// TIA Portal V17 export
// export: Created 2025-03-05T07:59:13.1679611Z, ExportSetting WithDefaults, DisplayName Totally Integrated Automation Portal, DisplayVersion V17 Update 8, DisplayName TIA Portal Openness, DisplayVersion V17 Update 8, DisplayName TIA Portal Version Control Interface, DisplayVersion V17, DisplayName SINAMICS Startdrive Advanced, DisplayVersion V17 SP2, DisplayName SINAMICS Startdrive G110M, G120, G120C, G120D, G120P, G115D, DisplayVersion V17 SP2, DisplayName SINAMICS Startdrive G130, G150, S120, S150, SINAMICS MV, S210, DisplayVersion V17 SP2, DisplayName STEP 7 Professional, DisplayVersion V17 Update 8, DisplayName SINUMERIK ONE STEP 7 Toolbox, DisplayVersion V17 Update 12, DisplayName SINUMERIK 840D sl STEP 7 Toolbox, DisplayVersion V17 Update 12, DisplayName STEP 7 Safety, DisplayVersion V17 Update 6, DisplayName WinCC Advanced, DisplayVersion V17 Update 8
FUNCTION "FC4001_FIXTURES_CALIBRATION" : Void   // FC4001, LAD
{ S7_Optimized_Access := 'TRUE' }
VERSION : 0.1
// stored: AutoNumber false, IsIECCheckEnabled false, SetENOAutomatically false, UDAEnableTagReadback false
BEGIN

REGION Network 1: FIXTURE 1 STATION 2 CALIBRATION DONE MEMORY
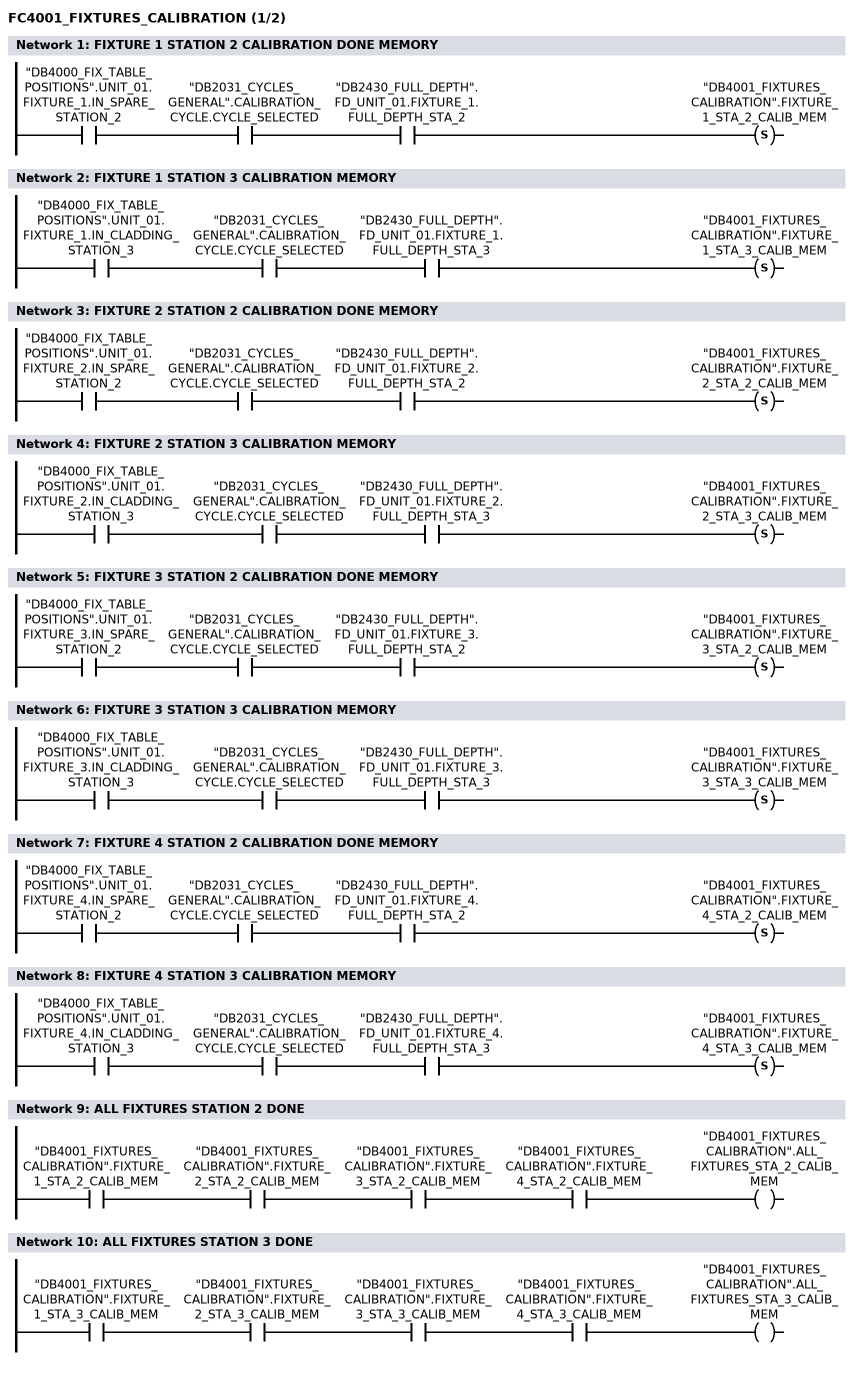
   RUNG wire#powerrail
      Contact( "DB4000_FIX_TABLE_POSITIONS".UNIT_01.FIXTURE_1.IN_SPARE_STATION_2 )
      Contact( "DB2031_CYCLES_GENERAL".CALIBRATION_CYCLE.CYCLE_SELECTED )
      Contact( "DB2430_FULL_DEPTH".FD_UNIT_01.FIXTURE_1.FULL_DEPTH_STA_2 )
      S_Coil( "DB4001_FIXTURES_CALIBRATION".FIXTURE_1_STA_2_CALIB_MEM )
   END_RUNG
   // the same network as SCL:
   IF "DB4000_FIX_TABLE_POSITIONS".UNIT_01.FIXTURE_1.IN_SPARE_STATION_2 AND "DB2031_CYCLES_GENERAL".CALIBRATION_CYCLE.CYCLE_SELECTED AND "DB2430_FULL_DEPTH".FD_UNIT_01.FIXTURE_1.FULL_DEPTH_STA_2 THEN
       "DB4001_FIXTURES_CALIBRATION".FIXTURE_1_STA_2_CALIB_MEM := TRUE;
   END_IF;
END_REGION

REGION Network 2: FIXTURE 1 STATION 3 CALIBRATION MEMORY
   RUNG wire#powerrail
      Contact( "DB4000_FIX_TABLE_POSITIONS".UNIT_01.FIXTURE_1.IN_CLADDING_STATION_3 )
      Contact( "DB2031_CYCLES_GENERAL".CALIBRATION_CYCLE.CYCLE_SELECTED )
      Contact( "DB2430_FULL_DEPTH".FD_UNIT_01.FIXTURE_1.FULL_DEPTH_STA_3 )
      S_Coil( "DB4001_FIXTURES_CALIBRATION".FIXTURE_1_STA_3_CALIB_MEM )
   END_RUNG
   // the same network as SCL:
   IF "DB4000_FIX_TABLE_POSITIONS".UNIT_01.FIXTURE_1.IN_CLADDING_STATION_3 AND "DB2031_CYCLES_GENERAL".CALIBRATION_CYCLE.CYCLE_SELECTED AND "DB2430_FULL_DEPTH".FD_UNIT_01.FIXTURE_1.FULL_DEPTH_STA_3 THEN
       "DB4001_FIXTURES_CALIBRATION".FIXTURE_1_STA_3_CALIB_MEM := TRUE;
   END_IF;
END_REGION

REGION Network 3: FIXTURE 2 STATION 2 CALIBRATION DONE MEMORY
   RUNG wire#powerrail
      Contact( "DB4000_FIX_TABLE_POSITIONS".UNIT_01.FIXTURE_2.IN_SPARE_STATION_2 )
      Contact( "DB2031_CYCLES_GENERAL".CALIBRATION_CYCLE.CYCLE_SELECTED )
      Contact( "DB2430_FULL_DEPTH".FD_UNIT_01.FIXTURE_2.FULL_DEPTH_STA_2 )
      S_Coil( "DB4001_FIXTURES_CALIBRATION".FIXTURE_2_STA_2_CALIB_MEM )
   END_RUNG
   // the same network as SCL:
   IF "DB4000_FIX_TABLE_POSITIONS".UNIT_01.FIXTURE_2.IN_SPARE_STATION_2 AND "DB2031_CYCLES_GENERAL".CALIBRATION_CYCLE.CYCLE_SELECTED AND "DB2430_FULL_DEPTH".FD_UNIT_01.FIXTURE_2.FULL_DEPTH_STA_2 THEN
       "DB4001_FIXTURES_CALIBRATION".FIXTURE_2_STA_2_CALIB_MEM := TRUE;
   END_IF;
END_REGION

REGION Network 4: FIXTURE 2 STATION 3 CALIBRATION MEMORY
   RUNG wire#powerrail
      Contact( "DB4000_FIX_TABLE_POSITIONS".UNIT_01.FIXTURE_2.IN_CLADDING_STATION_3 )
      Contact( "DB2031_CYCLES_GENERAL".CALIBRATION_CYCLE.CYCLE_SELECTED )
      Contact( "DB2430_FULL_DEPTH".FD_UNIT_01.FIXTURE_2.FULL_DEPTH_STA_3 )
      S_Coil( "DB4001_FIXTURES_CALIBRATION".FIXTURE_2_STA_3_CALIB_MEM )
   END_RUNG
   // the same network as SCL:
   IF "DB4000_FIX_TABLE_POSITIONS".UNIT_01.FIXTURE_2.IN_CLADDING_STATION_3 AND "DB2031_CYCLES_GENERAL".CALIBRATION_CYCLE.CYCLE_SELECTED AND "DB2430_FULL_DEPTH".FD_UNIT_01.FIXTURE_2.FULL_DEPTH_STA_3 THEN
       "DB4001_FIXTURES_CALIBRATION".FIXTURE_2_STA_3_CALIB_MEM := TRUE;
   END_IF;
END_REGION

REGION Network 5: FIXTURE 3 STATION 2 CALIBRATION DONE MEMORY
   RUNG wire#powerrail
      Contact( "DB4000_FIX_TABLE_POSITIONS".UNIT_01.FIXTURE_3.IN_SPARE_STATION_2 )
      Contact( "DB2031_CYCLES_GENERAL".CALIBRATION_CYCLE.CYCLE_SELECTED )
      Contact( "DB2430_FULL_DEPTH".FD_UNIT_01.FIXTURE_3.FULL_DEPTH_STA_2 )
      S_Coil( "DB4001_FIXTURES_CALIBRATION".FIXTURE_3_STA_2_CALIB_MEM )
   END_RUNG
   // the same network as SCL:
   IF "DB4000_FIX_TABLE_POSITIONS".UNIT_01.FIXTURE_3.IN_SPARE_STATION_2 AND "DB2031_CYCLES_GENERAL".CALIBRATION_CYCLE.CYCLE_SELECTED AND "DB2430_FULL_DEPTH".FD_UNIT_01.FIXTURE_3.FULL_DEPTH_STA_2 THEN
       "DB4001_FIXTURES_CALIBRATION".FIXTURE_3_STA_2_CALIB_MEM := TRUE;
   END_IF;
END_REGION

REGION Network 6: FIXTURE 3 STATION 3 CALIBRATION MEMORY
   RUNG wire#powerrail
      Contact( "DB4000_FIX_TABLE_POSITIONS".UNIT_01.FIXTURE_3.IN_CLADDING_STATION_3 )
      Contact( "DB2031_CYCLES_GENERAL".CALIBRATION_CYCLE.CYCLE_SELECTED )
      Contact( "DB2430_FULL_DEPTH".FD_UNIT_01.FIXTURE_3.FULL_DEPTH_STA_3 )
      S_Coil( "DB4001_FIXTURES_CALIBRATION".FIXTURE_3_STA_3_CALIB_MEM )
   END_RUNG
   // the same network as SCL:
   IF "DB4000_FIX_TABLE_POSITIONS".UNIT_01.FIXTURE_3.IN_CLADDING_STATION_3 AND "DB2031_CYCLES_GENERAL".CALIBRATION_CYCLE.CYCLE_SELECTED AND "DB2430_FULL_DEPTH".FD_UNIT_01.FIXTURE_3.FULL_DEPTH_STA_3 THEN
       "DB4001_FIXTURES_CALIBRATION".FIXTURE_3_STA_3_CALIB_MEM := TRUE;
   END_IF;
END_REGION

REGION Network 7: FIXTURE 4 STATION 2 CALIBRATION DONE MEMORY
   RUNG wire#powerrail
      Contact( "DB4000_FIX_TABLE_POSITIONS".UNIT_01.FIXTURE_4.IN_SPARE_STATION_2 )
      Contact( "DB2031_CYCLES_GENERAL".CALIBRATION_CYCLE.CYCLE_SELECTED )
      Contact( "DB2430_FULL_DEPTH".FD_UNIT_01.FIXTURE_4.FULL_DEPTH_STA_2 )
      S_Coil( "DB4001_FIXTURES_CALIBRATION".FIXTURE_4_STA_2_CALIB_MEM )
   END_RUNG
   // the same network as SCL:
   IF "DB4000_FIX_TABLE_POSITIONS".UNIT_01.FIXTURE_4.IN_SPARE_STATION_2 AND "DB2031_CYCLES_GENERAL".CALIBRATION_CYCLE.CYCLE_SELECTED AND "DB2430_FULL_DEPTH".FD_UNIT_01.FIXTURE_4.FULL_DEPTH_STA_2 THEN
       "DB4001_FIXTURES_CALIBRATION".FIXTURE_4_STA_2_CALIB_MEM := TRUE;
   END_IF;
END_REGION

REGION Network 8: FIXTURE 4 STATION 3 CALIBRATION MEMORY
   RUNG wire#powerrail
      Contact( "DB4000_FIX_TABLE_POSITIONS".UNIT_01.FIXTURE_4.IN_CLADDING_STATION_3 )
      Contact( "DB2031_CYCLES_GENERAL".CALIBRATION_CYCLE.CYCLE_SELECTED )
      Contact( "DB2430_FULL_DEPTH".FD_UNIT_01.FIXTURE_4.FULL_DEPTH_STA_3 )
      S_Coil( "DB4001_FIXTURES_CALIBRATION".FIXTURE_4_STA_3_CALIB_MEM )
   END_RUNG
   // the same network as SCL:
   IF "DB4000_FIX_TABLE_POSITIONS".UNIT_01.FIXTURE_4.IN_CLADDING_STATION_3 AND "DB2031_CYCLES_GENERAL".CALIBRATION_CYCLE.CYCLE_SELECTED AND "DB2430_FULL_DEPTH".FD_UNIT_01.FIXTURE_4.FULL_DEPTH_STA_3 THEN
       "DB4001_FIXTURES_CALIBRATION".FIXTURE_4_STA_3_CALIB_MEM := TRUE;
   END_IF;
END_REGION

REGION Network 9: ALL FIXTURES STATION 2 DONE
   RUNG wire#powerrail
      Contact( "DB4001_FIXTURES_CALIBRATION".FIXTURE_1_STA_2_CALIB_MEM )
      Contact( "DB4001_FIXTURES_CALIBRATION".FIXTURE_2_STA_2_CALIB_MEM )
      Contact( "DB4001_FIXTURES_CALIBRATION".FIXTURE_3_STA_2_CALIB_MEM )
      Contact( "DB4001_FIXTURES_CALIBRATION".FIXTURE_4_STA_2_CALIB_MEM )
      Coil( "DB4001_FIXTURES_CALIBRATION".ALL_FIXTURES_STA_2_CALIB_MEM )
   END_RUNG
   // the same network as SCL:
   "DB4001_FIXTURES_CALIBRATION".ALL_FIXTURES_STA_2_CALIB_MEM := "DB4001_FIXTURES_CALIBRATION".FIXTURE_1_STA_2_CALIB_MEM AND "DB4001_FIXTURES_CALIBRATION".FIXTURE_2_STA_2_CALIB_MEM AND "DB4001_FIXTURES_CALIBRATION".FIXTURE_3_STA_2_CALIB_MEM AND "DB4001_FIXTURES_CALIBRATION".FIXTURE_4_STA_2_CALIB_MEM;
END_REGION

REGION Network 10: ALL FIXTURES STATION 3 DONE
   RUNG wire#powerrail
      Contact( "DB4001_FIXTURES_CALIBRATION".FIXTURE_1_STA_3_CALIB_MEM )
      Contact( "DB4001_FIXTURES_CALIBRATION".FIXTURE_2_STA_3_CALIB_MEM )
      Contact( "DB4001_FIXTURES_CALIBRATION".FIXTURE_3_STA_3_CALIB_MEM )
      Contact( "DB4001_FIXTURES_CALIBRATION".FIXTURE_4_STA_3_CALIB_MEM )
      Coil( "DB4001_FIXTURES_CALIBRATION".ALL_FIXTURES_STA_3_CALIB_MEM )
   END_RUNG
   // the same network as SCL:
   "DB4001_FIXTURES_CALIBRATION".ALL_FIXTURES_STA_3_CALIB_MEM := "DB4001_FIXTURES_CALIBRATION".FIXTURE_1_STA_3_CALIB_MEM AND "DB4001_FIXTURES_CALIBRATION".FIXTURE_2_STA_3_CALIB_MEM AND "DB4001_FIXTURES_CALIBRATION".FIXTURE_3_STA_3_CALIB_MEM AND "DB4001_FIXTURES_CALIBRATION".FIXTURE_4_STA_3_CALIB_MEM;
END_REGION

REGION Network 11: ALL FIXTURES ALL STATIONS DONE
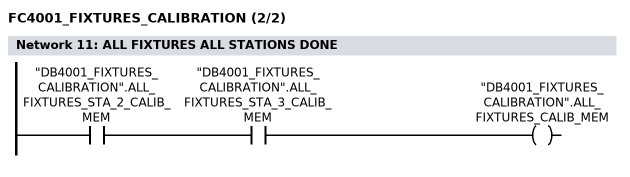
   RUNG wire#powerrail
      Contact( "DB4001_FIXTURES_CALIBRATION".ALL_FIXTURES_STA_2_CALIB_MEM )
      Contact( "DB4001_FIXTURES_CALIBRATION".ALL_FIXTURES_STA_3_CALIB_MEM )
      Coil( "DB4001_FIXTURES_CALIBRATION".ALL_FIXTURES_CALIB_MEM )
   END_RUNG
   // the same network as SCL:
   "DB4001_FIXTURES_CALIBRATION".ALL_FIXTURES_CALIB_MEM := "DB4001_FIXTURES_CALIBRATION".ALL_FIXTURES_STA_2_CALIB_MEM AND "DB4001_FIXTURES_CALIBRATION".ALL_FIXTURES_STA_3_CALIB_MEM;
END_REGION
END_FUNCTION
